// TIA Portal project "VtSys_4S" (V13)

(* hardware
DEVICE "S7300/ET200M-Station_1"  S7-300 station
   slot 0: "Profilschiene_0"  Rail  6ES7 390-1***0-0AA0
   slot 1: "PS 307 5A_1"  PS 307 5A  6ES7 307-1EA00-0AA0
   slot 2: "SIMATIC S7-300"  CPU 314C-2 PN/DP  6ES7 314-6EH04-0AB0  V3.3
      slot 2: "PROFINET-Schnittstelle_1"  PN-IO
         slot 1: "Port_1"  Port
         slot 2: "Port_2"  Port
      slot 5: "DI 24/DO 16_1"  DI24/DO16
      slot 6: "AI 5/AO 2_1"  AI5/AO2
      slot 7: "Zählen_1"  Counter
      slot 8: "Positionieren_1"  Positioning
   slot 4: "CP 343-2_1"  CP 343-2  6GK7 343-2AH01-0XA0  V3.1
*)

// ===== PLC "SIMATIC S7-300"  CPU 314C-2 PN/DP =====

VAR_GLOBAL   // PLC tag table "Standard-Variablentabelle"
   "Mx_Clock10Hz" AT %M100.0 : Bool;   // CPU clock memory-flag 0: f = 10 Hz / T = 0,1 s
   "Mx_Clock5Hz" AT %M100.1 : Bool;   // CPU clock memory-flag 1: f = 5 Hz / T = 0,2 s
   "Mx_Clock2,5Hz" AT %M100.2 : Bool;   // CPU clock memory-flag 2: f = 2,5 Hz / T = 0,4 s
   "Mx_Clock2Hz" AT %M100.3 : Bool;   // CPU clock memory-flag 3: f = 2 Hz / T = 0,5 s
   "Mx_Clock1,25Hz" AT %M100.4 : Bool;   // CPU clock memory-flag 4: f = 1,25 Hz / T = 0,8 s
   "Mx_Clock1Hz" AT %M100.5 : Bool;   // CPU clock memory-flag 5: f = 1 Hz / T = 1 s
   "Mx_Clock0,625Hz" AT %M100.6 : Bool;   // CPU clock memory-flag 6: f = 0,625 Hz / T = 1,6 s
   "Mx_Clock0,5Hz" AT %M100.7 : Bool;   // CPU clock memory-flag 7: f = 0,5 Hz / T = 2 s
   "Ix_S0_OFF" AT %I124.0 : Bool;   // Fan motors M1 to M4 off (NC)
   "Ix_F1(S1)_Overload_Fan1" AT %I124.1 : Bool;   // Overload relay F1, motor 1 (NC)
   "Ix_F2(S2)_Overload_Fan2" AT %I124.2 : Bool;   // Overload relay F2, motor 2 (NC)
   "Mx_Step1" AT %M10.0 : Bool;   // Grafcet G1, step-flag 1
   "Mx_Step2" AT %M10.1 : Bool;   // Grafcet G1, step-flag 2
   "Mx_Step20" AT %M10.2 : Bool;   // Grafcet G20, step-flag 20
   "Mx_Step30" AT %M10.3 : Bool;   // Grafcet G30, step-flag 30
   "Mx_StartingFlag" AT %M20.0 : Bool;   // Starting flag to activate the sequence (step 1)
   "Mx_PEdgeFlag_Step1" AT %M20.1 : Bool;   // Positive edge flag is activated when step 1 is activated
   "Mb_FlagByte10" AT %MB10 : Byte;   // Flag byte 10
   "Ix_F3(S3)_Overload_Fan3" AT %I124.3 : Bool;   // Overload relay F3, motor 3 (NC)
   "Ix_F4(S4)_Overload_Fan4" AT %I124.4 : Bool;   // Overload relay F4, motor 4 (NC)
   "Ix_S5_ON" AT %I124.5 : Bool;   // Fan motors M1 to M4 on
   "Qx_P-RD_TrafficLightRed" AT %Q124.0 : Bool;   // Traffic light red
   "Cx_VehicleCounter" AT %C1 : Counter;   // Counter to count the number of vehicles
   "Ix_B1_IncomingVehicles" AT %I124.6 : Bool;   // Sensor to detect incoming vehicles
   "Ix_B2_OutgoingVehicles" AT %I124.7 : Bool;   // Sensor to detect outgoing vehicles
   "Ix_S6_ResetCounter" AT %I125.0 : Bool;   // Reset vehicle counter
   "Mw_CV_WORD" AT %MW30 : Word;   // Count value in the format WORD
   "Mw_CV_INT" AT %MW32 : Int;   // Count value in the format INTEGER
   "Qx_P-YE_TrafficLightYellow" AT %Q124.1 : Bool;   // Traffic light yellow
   "Qx_P-GN_TrafficLightGreen" AT %Q124.2 : Bool;   // Traffic light green
   "Qx_Q1(P1)_Fan1" AT %Q125.0 : Bool;   // Fan motor 1 (main contactor and signal lamp)
   "Qx_Q2(P2)_Fan2" AT %Q125.1 : Bool;   // Fan motor 2 (main contactor and signal lamp)
   "Qx_Q3(P3)_Fan3" AT %Q125.2 : Bool;   // Fan motor 3 (main contactor and signal lamp)
   "Qx_Q4(P4)_Fan4" AT %Q125.3 : Bool;   // Fan motor 4 (main contactor and signal lamp)
   "Mx_LockVehicleCounter" AT %M10.7 : Bool;   // Lock the up counter
END_VAR

DATA_BLOCK "Fan Control_1"   // DB1
{ S7_Optimized_Access := 'FALSE' }
VERSION : 0.1
// stored: InstanceOfName Fan Control
"Fan Control"
BEGIN
END_DATA_BLOCK

DATA_BLOCK "Fan Control_2"   // DB2
{ S7_Optimized_Access := 'FALSE' }
VERSION : 0.1
// stored: InstanceOfName Fan Control
"Fan Control"
BEGIN
END_DATA_BLOCK

DATA_BLOCK "Fan Control_3"   // DB3
{ S7_Optimized_Access := 'FALSE' }
VERSION : 0.1
// stored: InstanceOfName Fan Control
"Fan Control"
BEGIN
END_DATA_BLOCK

DATA_BLOCK "Fan Control_4"   // DB4
{ S7_Optimized_Access := 'FALSE' }
VERSION : 0.1
// stored: InstanceOfName Fan Control
"Fan Control"
BEGIN
END_DATA_BLOCK

FUNCTION_BLOCK "Fan Control"   // FB1, FBD
{ S7_Optimized_Access := 'FALSE' }
VERSION : 0.1
   VAR_TEMP   // added for the SCL form of the ladder/FBD networks
      _w1 : Bool;
      _w2 : Bool;
   END_VAR
BEGIN

REGION Network 1
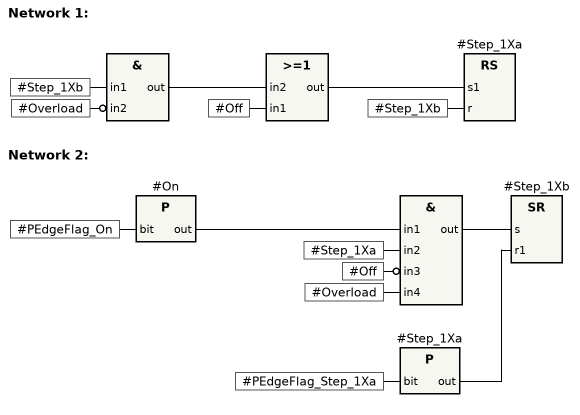
   IF #Step_1Xb THEN
       #Step_1Xa := FALSE;   // RS flip-flop
   END_IF;
   IF (#Step_1Xb AND NOT #Overload) OR #Off THEN #Step_1Xa := TRUE; END_IF;
END_REGION

REGION Network 2
   #_w1 := #On AND NOT #PEdgeFlag_On;   // rising edge of #On
   #PEdgeFlag_On := #On;
   #_w2 := #Step_1Xa AND NOT #PEdgeFlag_Step_1Xa;   // rising edge of #Step_1Xa
   #PEdgeFlag_Step_1Xa := #Step_1Xa;
   IF #_w1 AND #Step_1Xa AND NOT #Off AND #Overload THEN
       #Step_1Xb := TRUE;   // SR flip-flop
   END_IF;
   IF #_w2 THEN #Step_1Xb := FALSE; END_IF;
END_REGION
END_FUNCTION_BLOCK

FUNCTION "Main Switch" : Void   // FC1, FBD
{ S7_Optimized_Access := 'FALSE' }
VERSION : 0.1
   VAR_TEMP   // added for the SCL form of the ladder/FBD networks
      _w1 : Bool;
   END_VAR
BEGIN

REGION Network 1: Grafcet G1, step-flag 1
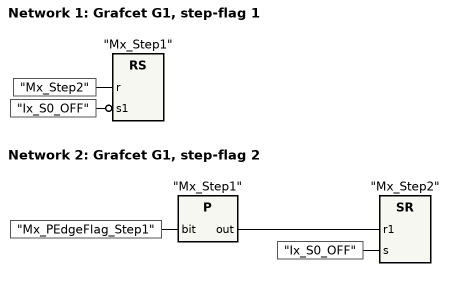
   IF "Mx_Step2" THEN
       "Mx_Step1" := FALSE;   // RS flip-flop
   END_IF;
   IF NOT "Ix_S0_OFF" THEN "Mx_Step1" := TRUE; END_IF;
END_REGION

REGION Network 2: Grafcet G1, step-flag 2
   #_w1 := "Mx_Step1" AND NOT "Mx_PEdgeFlag_Step1";   // rising edge of "Mx_Step1"
   "Mx_PEdgeFlag_Step1" := "Mx_Step1";
   IF "Ix_S0_OFF" THEN
       "Mx_Step2" := TRUE;   // SR flip-flop
   END_IF;
   IF #_w1 THEN "Mx_Step2" := FALSE; END_IF;
END_REGION
END_FUNCTION

FUNCTION "Actions" : Void   // FC2, FBD
{ S7_Optimized_Access := 'FALSE' }
VERSION : 0.1
BEGIN

REGION Network 1: Fan controll 1
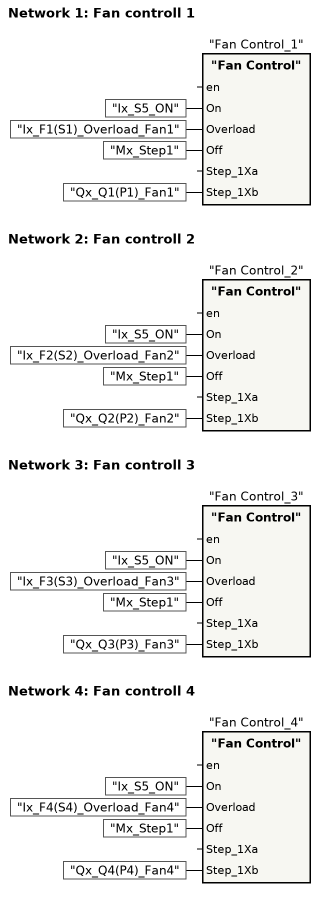
   "Fan Control_1"(On := "Ix_S5_ON",   // "Fan Control"
                   Overload := "Ix_F1(S1)_Overload_Fan1",
                   Off := "Mx_Step1",
                   Step_1Xb := "Qx_Q1(P1)_Fan1");
END_REGION

REGION Network 2: Fan controll 2
   "Fan Control_2"(On := "Ix_S5_ON",   // "Fan Control"
                   Overload := "Ix_F2(S2)_Overload_Fan2",
                   Off := "Mx_Step1",
                   Step_1Xb := "Qx_Q2(P2)_Fan2");
END_REGION

REGION Network 3: Fan controll 3
   "Fan Control_3"(On := "Ix_S5_ON",   // "Fan Control"
                   Overload := "Ix_F3(S3)_Overload_Fan3",
                   Off := "Mx_Step1",
                   Step_1Xb := "Qx_Q3(P3)_Fan3");
END_REGION

REGION Network 4: Fan controll 4
   "Fan Control_4"(On := "Ix_S5_ON",   // "Fan Control"
                   Overload := "Ix_F4(S4)_Overload_Fan4",
                   Off := "Mx_Step1",
                   Step_1Xb := "Qx_Q4(P4)_Fan4");
END_REGION
END_FUNCTION

FUNCTION "Trafic Light" : Void   // FC20, FBD
{ S7_Optimized_Access := 'FALSE' }
VERSION : 0.1
BEGIN

REGION Network 1: Trafic light red
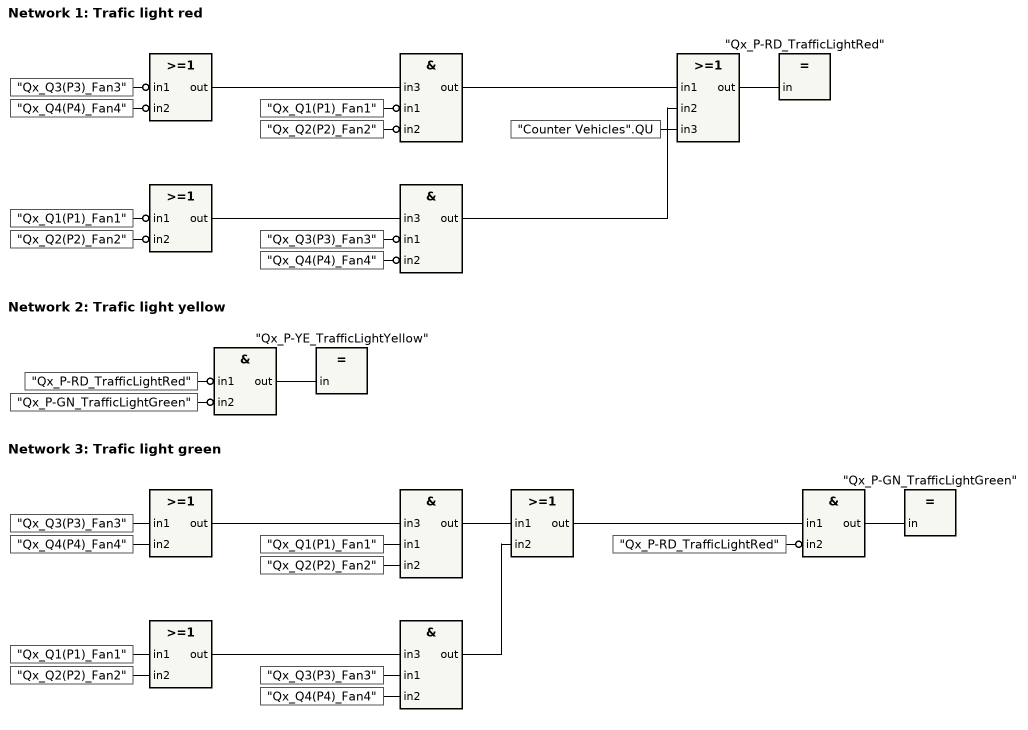
   "Qx_P-RD_TrafficLightRed" := ((NOT "Qx_Q3(P3)_Fan3" OR NOT "Qx_Q4(P4)_Fan4") AND NOT "Qx_Q1(P1)_Fan1" AND NOT "Qx_Q2(P2)_Fan2") OR ((NOT "Qx_Q1(P1)_Fan1" OR NOT "Qx_Q2(P2)_Fan2") AND NOT "Qx_Q3(P3)_Fan3" AND NOT "Qx_Q4(P4)_Fan4") OR "Counter Vehicles".QU;
END_REGION

REGION Network 2: Trafic light yellow
   "Qx_P-YE_TrafficLightYellow" := NOT "Qx_P-RD_TrafficLightRed" AND NOT "Qx_P-GN_TrafficLightGreen";
END_REGION

REGION Network 3: Trafic light green
   "Qx_P-GN_TrafficLightGreen" := ((("Qx_Q3(P3)_Fan3" OR "Qx_Q4(P4)_Fan4") AND "Qx_Q1(P1)_Fan1" AND "Qx_Q2(P2)_Fan2") OR (("Qx_Q1(P1)_Fan1" OR "Qx_Q2(P2)_Fan2") AND "Qx_Q3(P3)_Fan3" AND "Qx_Q4(P4)_Fan4")) AND NOT "Qx_P-RD_TrafficLightRed";
END_REGION
END_FUNCTION

FUNCTION "Vehicle Counter" : Void   // FC30, FBD
{ S7_Optimized_Access := 'FALSE' }
VERSION : 0.1
BEGIN

REGION Network 1: Couting the vehicles
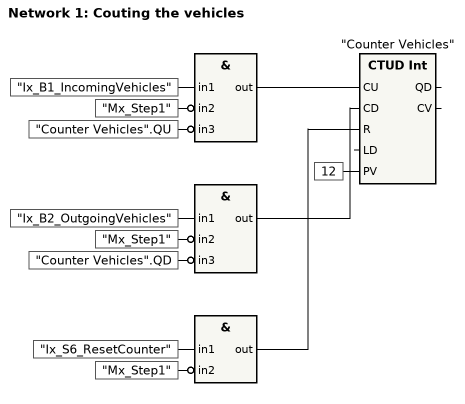
   "Counter Vehicles".CTUD(CU := "Ix_B1_IncomingVehicles" AND NOT "Mx_Step1" AND NOT "Counter Vehicles".QU,
                           CD := "Ix_B2_OutgoingVehicles" AND NOT "Mx_Step1" AND NOT "Counter Vehicles".QD,
                           R := "Ix_S6_ResetCounter" AND NOT "Mx_Step1",
                           PV := 12);
END_REGION
END_FUNCTION

ORGANIZATION_BLOCK "Main"   // OB1, FBD
TITLE = "Main Program Sweep (Cycle)"
{ S7_Optimized_Access := 'FALSE' }
VERSION : 0.1
// Organisation block OB1 is executed cyclically
BEGIN

REGION Network 1: Call the function diagram block G1 ("main switch")
   // Programming of the function diagram (Grafcet)
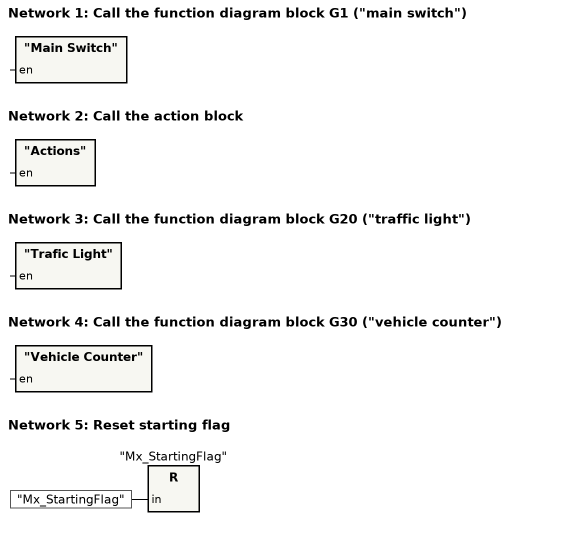
   "Main Switch"();
END_REGION

REGION Network 2: Call the action block
   // Programming of the actions
   "Actions"();
END_REGION

REGION Network 3: Call the function diagram block G20 ("traffic light")
   // Programming of the function diagram (Grafcet)
   "Trafic Light"();
END_REGION

REGION Network 4: Call the function diagram block G30 ("vehicle counter")
   // Programming of the function diagram (Grafcet)
   "Vehicle Counter"();
END_REGION

REGION Network 5: Reset starting flag
   IF "Mx_StartingFlag" THEN "Mx_StartingFlag" := FALSE; END_IF;
END_REGION
END_ORGANIZATION_BLOCK

ORGANIZATION_BLOCK "COMPLETE RESTART"   // OB100, FBD
TITLE = "Complete Restart"
{ S7_Optimized_Access := 'FALSE' }
VERSION : 0.1
BEGIN

REGION Network 1: Reset Flagbyte 10
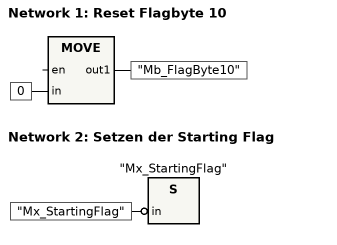
   "Mb_FlagByte10" := 0;
END_REGION

REGION Network 2: Setzen der Starting Flag
   IF NOT "Mx_StartingFlag" THEN "Mx_StartingFlag" := TRUE; END_IF;
END_REGION
END_ORGANIZATION_BLOCK